KUKA KRL data list: global_eki.dat

&ACCESS RVP
&REL 48
defdat global_eki public
   global real axis_set_velocity
enddat
